KUKA KRL program: makrosps5.src

&ACCESS RV
&PARAM TEMPLATE = C:\KRC\Roboter\Template\makrospsvorgabe.src
&PARAM EDITMASK = MakroSPS5
&PARAM TPVW_VERSION=8.3.18
DEF MAKROSPS5 ( )
; FOLD Makro Anfang;%{PSE} %MKUKATPVW
SPS_N=-1
; ENDFOLD
; FOLD ;%{H}
END
; ENDFOLD
